{attribute addProperty BoxType "EPP1111-0000-0016"}
{attribute addProperty Id "IDAT %I*UINT162"}
{attribute addProperty CRC "2432610056"}
{attribute addProperty SizeInBites "16"}
{attribute addProperty SizeInBytes "2"}
TYPE ID_Inputs_90FEAF08 :
STRUCT
	{attribute addProperty Name "ID"}
	ID AT %I* : UINT;
END_STRUCT
END_TYPE

(* stored: Version 1.2.0.0, ProductVersion 3.1.4024.9
   DUT ID_Inputs_90FEAF08: Id {c2afd733-2a74-45ab-b796-20b1b884192d} *)
